// Contains varias TwinCAT Runtime datatypes for tcads-rs's DataTypeDevice
PROGRAM P_DataTypesExample
VAR
	fbCalc 						: FB_EmptyWithRPC;
	// Interfaces
	
	ipEmpty 					: I_Empty;
	ipEmptyWithExtends 			: I_EmptyWithExtends;
	ipWithProps					: I_WithProps;
	ipWithMethods				: I_WithMethods;
	ipWithMethodPropsAndExtends : I_WithMethodsPropsAndExtends;
	ipWithRPC					: I_WithRPC;
	
	// Function Blocks
	
	fbEmpty 					: FB_Empty;
	fbEmptyWithExtends 			: FB_EmptyWithExtends;
	fbEmptyWithEmptyImpl		: FB_EmptyWithEmptyImpl;
	fbWithFields				: FB_WithFields;
	fbEmptyWithRPC 				: FB_EmptyWithRPC;
	fbEmptyWithImplRPC 			: FB_EmptyWithImplRPC;
	
	// Structs
	
	stEmpty						: ST_Empty;
	STEmptyAlias				: T_STEmptyAlias;	
END_VAR

END_PROGRAM

(* stored: Version 1.1.0.1, ProductVersion 3.1.4024.15
   POU P_DataTypesExample: Id {e2674363-e098-4b6d-9106-aea4ebc035fd}, SpecialFunc None *)
